PROGRAM MAIN
VAR
	// OPC UA mapper for cell
	{attribute 'OPC.UA.DA':='1'}
	Bridge					: FB_OPC_Cell_Unit_4;

// Cell handling, PackML etc.
	fbUnit4					: FB_Cell_Unit_4;

// Log to file
	fbLogToFile				: FB_LogToFile;
	
//	LicenseState	AT %I*	: UINT;
	bInitDone 				: BOOL;
	
END_VAR


M_Init();

// Cell handling
fbUnit4(stModeStateIn := Bridge.Input.Cell.ModeState, 
		stModeStateOut := Bridge.Output.Cell.ModeState,
		stOEE := Bridge.Output.Cell.OEE,
		stErrorWarning := Bridge.Output.Cell.ErrorWarning,
		bResetEStop:= Bridge.P_bResetEStop,
		bLockDoor:= Bridge.P_bLockDoors, 
		bUnlockDoor:= Bridge.P_bUnlockDoors, 
		bCellLight:= Bridge.P_bCellLight,
		iHeartBeatFromMES:= Bridge.P_iHeartBeat,
		Input := Bridge.Input,		// Bridge Data Inputs
		Output := Bridge.Output, 	// Bridge Data Outputs
		bModeChangeInProcess=> 	);
		

// OPC handling
	// OPC handling
	Bridge.P_bEStop := fbUnit4.bEStopOK; 
	Bridge.P_bDoors := fbUnit4.bDoorsOK;
	Bridge.P_bCellLight := fbUnit4.bCellLightOn;
	Bridge.P_rPLCCPUTemp := fbUnit4.rCPUTemp;
	Bridge.P_rSafetyCPUTemp := fbUnit4.rSafetyTemp;
	Bridge.P_sPLCSerial := fbUnit4.sSerialIPC;
	Bridge.P_sPLCMBSerial := fbUnit4.sSerialMB;
	Bridge.P_bStationCommOK := NOT fbUnit4.bStationCommError;
	Bridge.P_iHeartBeat := fbUnit4.iHeartBeatToMES;
	Bridge.P_rOSCPULoad := fbUnit4.rCPULoad;
	Bridge.P_rPLCCPULoad := fbUnit4.rCPULoadPLC;
	Bridge.P_rCPUFrequency := fbUnit4.rCPUFrequency;
	Bridge();

//File logging
fbLocalTime(
	sNetID:= '', 
	bEnable:= TRUE, 
	dwCycle:= 5, 
	dwOpt:= 0, 
	tTimeout:=DEFAULT_ADS_TIMEOUT );	
	
fbLogToFile(Busy=> );

METHOD M_Init : BOOL
VAR_INPUT
END_VAR
// Init
IF (NOT bInitDone) THEN

	bInitDone := TRUE;
END_IF
END_METHOD

END_PROGRAM

(* stored: Version 1.1.0.1, ProductVersion 3.1.4024.5
   POU MAIN: Id {e099f760-829f-42a0-bf37-df04f387259b}, SpecialFunc None
   Method M_Init: Id {e826824d-1859-4451-a7c9-63865682eeed} *)
